// TIA Portal V19 export
ORGANIZATION_BLOCK "PID_Control"   // OB30, FBD, CyclicInterrupt
{ S7_Optimized_Access := 'TRUE' }
// stored: SetENOAutomatically false
   VAR_INPUT
      Initial_Call : Bool;   // Initial call of this OB
      Event_Count : Int;   // Events discarded
   END_VAR
BEGIN

REGION Network 1
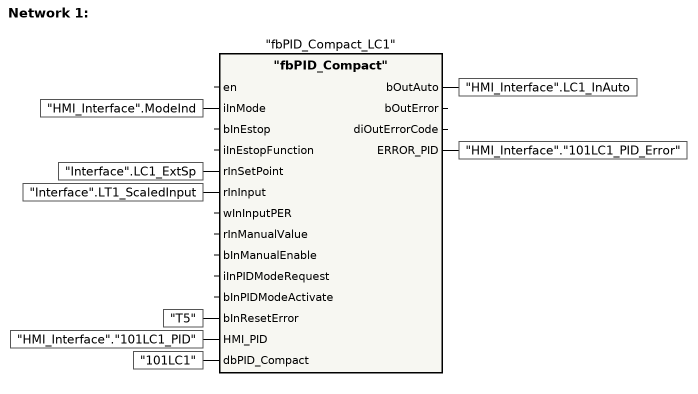
   "fbPID_Compact_LC1"(iInMode := "HMI_Interface".ModeInd,   // "fbPID_Compact"
                       rInSetPoint := "Interface".LC1_ExtSp,
                       rInInput := "Interface".LT1_ScaledInput,
                       bInResetError := "T5",
                       HMI_PID := "HMI_Interface"."101LC1_PID",
                       dbPID_Compact := "101LC1",
                       bOutAuto => "HMI_Interface".LC1_InAuto,
                       ERROR_PID => "HMI_Interface"."101LC1_PID_Error");
END_REGION
END_ORGANIZATION_BLOCK
